FUNCTION_BLOCK Sequencer_Test EXTENDS FB_TestSuite
VAR_INPUT
END_VAR
VAR_OUTPUT
END_VAR
VAR
END_VAR

// Copyright (c) 2024 Loupe (https://loupe.team), provided under the MIT License.

OnAbort();
OnEntry();
CurrentAndRequestStep();

METHOD CurrentAndRequestStep
VAR
    sequencer : Sequencer(0);
    Command : PLCopenCommand();
    step : UDINT;
END_VAR
// Copyright (c) 2024 Loupe (https://loupe.team), provided under the MIT License.

(*STweep.Disable*)

TEST('CurrentAndRequestStep');
	AssertEquals_UDINT(Expected := 0, Actual := sequencer.CurrentStep, Message := 'Current step shall default to 0');
	
	step := 2;
	sequencer.RequestStep(step);
	AssertEquals_UDINT(Expected := step, Actual := sequencer.CurrentStep, Message := 'Current step expected to be updated');
	
	step := 3;
	sequencer.RequestStepClear(step);
	AssertEquals_UDINT(Expected := step, Actual := sequencer.CurrentStep, Message := 'Current step expected to be updated');
TEST_FINISHED();
END_METHOD

METHOD OnAbort
VAR
    sequencer : Sequencer(0);
    outputVal : BOOL;
END_VAR
// Copyright (c) 2024 Loupe (https://loupe.team), provided under the MIT License.

(*STweep.Disable*)

TEST('SequenceOnAbort');
	sequencer.RequestStep(1);
	sequencer.SequenceAbort(0, 'Error message');
	sequencer.Run();
	outputVal := sequencer.OnAbort(1);
	AssertTrue(Condition := outputVal, Message := 'Abort should be true');
TEST_FINISHED();
END_METHOD

METHOD OnEntry
VAR_INPUT
END_VAR

VAR
    sequencer : Sequencer(0);
    outputVal : BOOL;
END_VAR
// Copyright (c) 2024 Loupe (https://loupe.team), provided under the MIT License.

(*STweep.Disable*)

TEST('OnEntry');
	
	sequencer.StartSequence();
	sequencer.DoStep();
	AssertTrue(Condition := sequencer.onEntry(), Message := 'onEntry should evaluate TRUE on first pass through a new step');
	sequencer.DoStep();
	AssertFalse(Condition := sequencer.onEntry(), Message := 'onEntry should evaluate FALSE on second pass');
	
TEST_FINISHED();
END_METHOD

METHOD OnError
VAR
    sequencer : Sequencer(0);
    outputVal : BOOL;
END_VAR
// Copyright (c) 2024 Loupe (https://loupe.team), provided under the MIT License.

(*STweep.Disable*)

TEST('SequenceOnError');
	sequencer.RequestStep(1);
	sequencer.SequenceError(0, 'Test Error');
	sequencer.Run();
	outputVal := sequencer.OnError(1);
	AssertTrue(Condition := outputVal, Message := 'Error should be true');
TEST_FINISHED();
END_METHOD

METHOD OnSuccess
VAR_INPUT
    sequencer : Sequencer(0);
END_VAR
// Copyright (c) 2024 Loupe (https://loupe.team), provided under the MIT License.

(*STweep.Disable*)

TEST('OnSuccess');

	//sequencer.i_sequence.activeTasks
	// next step negative
	//sequencer.setNextStep(-1);
	//sequencer.onSuccess(-1);
	
	// next step >= 0


TEST_FINISHED();
END_METHOD

METHOD Start
VAR
    sequencer : Sequencer(0);
    output : BOOL;
END_VAR
// Copyright (c) 2024 Loupe (https://loupe.team), provided under the MIT License.

(*STweep.Disable*)

TEST('Start');
	// activeTasks.Start) = 0
	// TODO
	
	//output := sequencer.i_sequence.startStep
	
	
TEST_FINISHED();
END_METHOD

END_FUNCTION_BLOCK

(* stored: Version 1.1.0.1
   POU Sequencer_Test: Id {5528d32b-0dad-48bc-b63b-5f76dadd2ea9}, SpecialFunc None
   Method CurrentAndRequestStep: Id {00c73c39-e570-45cb-8831-bed7304ddd26}
   Method OnAbort: Id {756190d0-8aa4-4061-8aca-7e61a0ad15cd}
   Method OnEntry: Id {3a0279ba-27ed-47d6-a39c-8c9f7c30b3c2}
   Method OnError: Id {ceefdcc0-adb1-4ad8-928a-8e1e77a9bfee}
   Method OnSuccess: Id {6a55c547-d864-42a2-86db-036e6aa1ad13}
   Method Start: Id {3d524a28-168c-402c-a8b1-706368e2797f} *)
